PROGRAM PRG_TEST
VAR
	fbSum_Test : FB_Sum_Test;
END_VAR

TcUnit.RUN();

END_PROGRAM

(* stored: Version 1.1.0.1, ProductVersion 3.1.4022.16
   POU PRG_TEST: Id {5e8cc903-e536-40be-a096-d6b305fbb618}, SpecialFunc None *)
